(* IEC 61131-3 sources: myCodes/Stone/07.02.2022 - OOPs Approach/MPx_One_New/Mpx_One_Source_Code/MPx_One/3. USHPXMPX010A1/USHPXMPX010A1/[8c990d04-4ef8-4ca1-9757-e845a4517aeb]/Application, 12 files *)

(* ---- 010_GeneralMng.st ---- *)
USING System.UI;
USING System;
USING System.Timer;
USING System.Serial;
USING System.NVRAM;
USING System.Logs;
USING Libs.Blackout;
USING Libs.Logics;
USING System.Math;
USING System.Text;
USING libs.GenericFunctionMng;

{IF DEF(MPX_LOGS)}
(* ONLY FOR DEBUG *)
VAR_GLOBAL
	LogsBuffer : ARRAY [0..1024] OF BYTE;
    myStrDebugCarel : STRING;
END_VAR
(* -------------- *)
{ENDIF}

VAR_GLOBAL
    (**Detect restarts of MPXone application*)
    powerUp : BOOL;
    (**Flag for recognize that a defrost was performed*)
    DfrPerformed : BOOL;
    (**flag for save sw_version after RetainRestoreDefault()*)
    SW_Update    : BOOL;
    (* Backup BMS Configuration fo upgrade SW  ------*)
    BMS_Addr_bkp : USINT;
    BMS_Baud_bkp : USINT;
    BMS_Conf_bkp : USINT;
    BMS_Prot_bkp : BOOL;
END_VAR

VAR_GLOBAL RETAIN
    (**Number of restrts of MPXone application *)
    RestartsCounter : UINT;
END_VAR

VAR_GLOBAL PERSISTENT
    (**Start for periodic log: hour*)
    {METADATA MAX_VAL 23}
    {METADATA MIN_VAL 0}
    {ATTRIBUTE UOM HOUR}
    StartLog_Hour : USINT (0..23) := 0;
    (**Start for periodic log: minute*)
    {METADATA MAX_VAL 59}
    {METADATA MIN_VAL 0}
    {ATTRIBUTE UOM MINUTE}
    StartLog_Min : USINT (0..59) := 0;

    StartLog_DT : DATE_AND_TIME;
END_VAR

NAMESPACE LibraryNamespaceAndVersion

PROGRAM GeneralMng

    VAR
        BMS_BaudPrec, BMS_ConfPrec, BMS_AddrPrec : USINT;
        FB_BaudPrec : USINT;

        FirsCheckBlackout : BOOL := FALSE;
        BlackoutCtl : Blackout;
        MyLastOffDate : DATE_AND_TIME;
        NVRAM_Array : DWORD;
        myPwrOffDate_NVRAM_BLKO : UDINT;

        CngCnfRT                : RF_TRIG;
        R_Trig_enNFC : R_TRIG;

        TON_WAIT_DOWNLOAD : TON;

        FirstRun : BOOL := TRUE;

        prevZoneHmi : BOOL;
        pCOType, boardType, machineType, hwCode : UINT;

        SPV_DT : DT;
        prevSPV_DT : DT := DATE_AND_TIME#2017-01-01-00:00:00;
        DisSpvUpdF_APP : BOOL;

        cfgId : SINT;
        cfgOk : BOOL;
        {IF NOT DEF(MPXONE_BASIC)}
        cfgName : STRING[16];
        {ELSE}
        cfgName : STRING[4];
        {ENDIF}
        UniqueId : LWORD;
    END_VAR

    VAR_TEMP
        ProdCode_HwID : USINT;
        ProdCode_ProdVers : USINT;
        tmp_Startlog : DateTime;
        tmp_CurrTime : DateTime;
        lastDfrTime_DWORD : DWORD;
        swVersion_tmp           : UINT;
    END_VAR

    {REGION HARDWARE INFO}
    GetHardwareDescription(HwDesc);
    GetModel(pCOType, boardType, machineType, hwCode);
    GetProductInfo(Product_Info);

    IF firstCycle THEN
        UniqueId := TO_LWORD(GetUniqueId());
        Split_UniqueId(UniqueId, UniqueID_SPV);

        {IF DEF(MPXONE_ADVANCED)}
        PwrSupplyFailure := FALSE;
        uConfig[9].mode_sel := 0; // U9 set as analog input to manageultracap control
        {ENDIF}

    END_IF;

    IF Product_Info.ProductCode <> '' THEN
        ProdCode_HwID := TO_USINT(MID(Product_Info.ProductCode, 2, 10));
        isPanelVersion := (ProdCode_HwID >= 5) AND (ProdCode_HwID <= 8);
        ProdCode_ProdVers := TO_USINT(MID(Product_Info.ProductCode, 1, 6));
        isCustomBasicRU := (ProdCode_ProdVers < 3) AND (ProdCode_HwID = 5);
        isProdBasicVersion := (ProdCode_ProdVers <= 4) AND (ProdCode_HwID <= 6);
    ELSE
        isPanelVersion := FALSE;
    END_IF;

    IF isCustomBasicRU THEN
        Ain_Types.Group1 := 1;
    END_IF;
    {ENDREGION}

    {REGION RESET TO DEFAULT IF SW VERSION IS DIFFERET OR MANUAL RESET}
                // Compose version variable for BMS and for reeset for update SW
    swVersion_tmp := __PROJ_VER_MAJOR__ * 1000 + __PROJ_VER_MINOR__ * 100 + __PROJ_VER_BUILD__;

    IF SW_Update THEN                   // at restart after RetainRestoreDefault() (below)
        swVersion := swVersion_tmp;     // save SW version
        SW_Update := FALSE;             // Stop reset time

            //Restore BMS settings only on change version (NOT on Manual Default request)
        IF NOT ResCarelSets THEN
            BMS_Addr :=BMS_Addr_bkp;
            BMS_Baud :=BMS_Baud_bkp;
            BMS_Conf :=BMS_Conf_bkp;
            BMS_Prot :=BMS_Prot_bkp;
        END_IF;

        DispMngInst.StartSync(DownloadDir#ACUtoHMI, FALSE); //Force param from ACU to NFC
        //RetainForceBackup();
        ResCarelSets := FALSE;
    END_IF;
    IF (swVersion <> swVersion_tmp AND NOT(SW_Update)) OR ResCarelSets THEN
        // Backup BMS configuration only
        BMS_Addr_bkp :=BMS_Addr;
        BMS_Baud_bkp :=BMS_Baud;
        BMS_Conf_bkp :=BMS_Conf;
        BMS_Prot_bkp :=BMS_Prot;
        RetainRestoreDefault(); //keep one program loop to be executed
        SW_Update    := TRUE;
    END_IF;
    {ENDREGION}

    {REGION Set DEFAULT values for analog input channels}

    // wiz done from Applica
    // for wiz done from HMI see: WIZ_ENDPRG.st
    IF WizDone AND WizProgress THEN
        WizDone_Action();
    END_IF;
    {ENDREGION}

    {REGION RESTART COUNTER}
    IF NOT powerUp THEN
        //poerUp := FALSE in PROGRAM OutputsMng
        RestartsCounter     := RestartsCounter + 1;
        LogsEventsCounter   := LogsEventsCounter + 1;
    END_IF;
    {ENDREGION}

    {REGION NFC and DISPLAY CHANGE management}
    R_Trig_enNFC(CLK := EnNfc);
    IF EnNfc THEN //AND NOT firstCycle THEN
        //DispMngInst.Check(isPanelVersion, IsCommissioningToolPresent() OR NOT(MasterOnlineTON.Q));
        IF NOT R_Trig_enNFC.Q OR NOT powerUp THEN
            DispMngInst.Check(FALSE, IsCommissioningToolPresent() OR NOT(MasterOnlineTON.Q));
        ELSE
            DispMngInst.StartSync(DownloadDir#ACUtoHMI, R_Trig_enNFC.Q);
        END_IF;

        //forcing parameter values from ACU to HMI in case of display change
        IF DispMngInst.isWaitingForUser() THEN
            NewDispPrompt := FALSE;
            DispMngInst.StartSync(DownloadDir#ACUtoHMI, FALSE);
        END_IF;
    END_IF;
    {ENDREGION}

    {IF DEF(NO_SEV_SUPPORT)}
	OneRow.Init();
	OneRow.Read();
    {ENDIF}

    // Find related compilation DEFINES
    {IF DEF(MPXONE_BASIC)}
    isBasic := TRUE;
    isMedium := FALSE;
    isAdvanced := FALSE;
    {ENDIF}

    {IF DEF(MPXONE_MEDIUM)}
    isBasic := TRUE;
    isMedium := TRUE;
    isAdvanced := FALSE;
    {ENDIF}

    {IF DEF(MPXONE_ADVANCED)}
    isBasic := TRUE;
    isMedium := TRUE;
    isAdvanced := TRUE;
    {ENDIF}

    {REGION CHANGE BMS SETTINGS}

    SpvTable.SerialPort.Settings.Channel := Serial_Channel#BMS1;
    (*change of BMS supervisor baudrate*)
    SpvTable.SerialPort.Settings.Speed := SetSerialSpeed(BMS_Baud);

    (*change of BMS supervisor settings*)
    SpvTable.SerialPort.Settings.Bits := 8;
    IF BMS_Conf > 5 THEN
        BMS_Conf := 0;
    END_IF;
    CASE BMS_Conf OF
        0:
            SpvTable.SerialPort.Settings.Parity := Serial_Parity#None;
            SpvTable.SerialPort.Settings.Stops := 1;
            (*8 NONE 1*)

        1:
            SpvTable.SerialPort.Settings.Parity := Serial_Parity#None;
            SpvTable.SerialPort.Settings.Stops := 2;
            (*8 NONE 2*)

        2:
            SpvTable.SerialPort.Settings.Parity := Serial_Parity#Even;
            SpvTable.SerialPort.Settings.Stops := 1;
            (*8 EVEN 1*)

        3:
            SpvTable.SerialPort.Settings.Parity := Serial_Parity#Even;
            SpvTable.SerialPort.Settings.Stops := 2;
            (*8 EVEN 2*)

        4:
            SpvTable.SerialPort.Settings.Parity := Serial_Parity#Odd;
            SpvTable.SerialPort.Settings.Stops := 1;
            (*8 ODD 1*)

        5:
            SpvTable.SerialPort.Settings.Parity := Serial_Parity#Odd;
            SpvTable.SerialPort.Settings.Stops := 2;
            (*8 ODD 2*)
    END_CASE;

    // Carel protocol works only at 19200 8n2
    IF NOT BMS_Prot AND ( BMS_Baud <> 4 OR BMS_Conf <> 1 ) THEN
        BMS_Baud := 4;
        BMS_Conf := 1;
    END_IF;

    (*change setting of supervisor port, just in case of modifications*)
    IF BMS_Baud <> BMS_BaudPrec OR BMS_Conf <> BMS_ConfPrec OR BMS_Addr <> BMS_AddrPrec THEN
        (* Set ID to allow STone communication *)
        SetModbusDebugID(BMS_Addr, SpvTable.serialPort.Settings.Channel);
        (* Adjust settings *)
        SerialChangeSettings(SpvTable.serialPort.Settings);

        IF BMS_Prot THEN
            MB_Slave.ChangeIdent(BMS_Addr);
        END_IF;

        BMS_BaudPrec := BMS_Baud;
        BMS_ConfPrec := BMS_Conf;
        BMS_AddrPrec := BMS_Addr;

        // Set the same settings for BMS port on Default app (In case of FW ugrade the device will be reachable with the same settings)
        SaveIdePortSettings(SpvTable.SerialPort.Settings.Channel, SpvTable.SerialPort.Settings.Speed,
            SpvTable.SerialPort.Settings.Bits, SpvTable.SerialPort.Settings.Parity, SpvTable.SerialPort.Settings.Stops, BMS_Addr);
    END_IF;

    IF FB_Baud <> FB_BaudPrec OR Fieldbus.SerialSettings.Speed <> SetSerialSpeed(FB_Baud) THEN

        Fieldbus.SerialSettings.Speed := SetSerialSpeed(FB_Baud);
        SerialChangeSettings(Fieldbus.SerialSettings);
        //Fieldbus.ChangeSettings();

        FB_BaudPrec := FB_Baud;
    END_IF;

    IF ZoneHMI THEN
        SpvTable.Info.Zone := System.Globalization.Imperial;
    ELSE
        SpvTable.Info.Zone := System.Globalization.SI;
    END_IF;

    IF ZoneHMI <> prevZoneHmi THEN
        prevZoneHmi := ZoneHMI;
        ChangedUoM := TRUE;
    ELSE
        ChangedUoM := FALSE;
    END_IF;

    Libs.SPV_Gateway_HPX.InitProtocols();

    IF WizDone AND NOT SlvUpdFW THEN

        SpvTable.Read(ChangedUoM, BMS_Prot);
        FieldBus.Read();
        {IF NOT DEF(NO_MPXONE_REPEATER)}
        mpxRepeater.Init(198, repeaterConfig);
        mpxRepeater.Check(HmiRemSel > 0);
        {ENDIF}
    END_IF;

    {ENDREGION }

    {REGION RTC WRITE}

    (*sets the time from app through NFC*)
    IF ToggleSetTimeAPP THEN

        SetTime(DateTimeToSet);
        SetTimeZone(Posix);

        // Avoid unexpected defrost changing RTC time
        GetLocalTime(CurrDateTime);
        //DfrStartedDT := CurrDateTime;

        ToggleSetTimeAPP := FALSE;
        //DisSpvUpdF := TRUE;
        DisSpvUpdF_APP := TRUE;

        // Reset alarm if any
        Alarms.Al.Al_RTC.Info.Trigger := FALSE;
    END_IF;

    // Update SPV Variables
    SPV_DT := CONCAT_DT(TO_UINT(SPV_Year) + 2000, TO_UINT(SPV_Month), TO_UINT(SPV_Day), TO_UINT(SPV_Hour), TO_UINT(SPV_Min), 0, 0);
    IF SPV_DT <> prevSPV_DT AND NOT FirstRun THEN

        // SPV has updated date/time of controller
        SetLocalTime(SPV_DT);

        // Avoid unexpected defrost changing RTC time
        GetLocalTime(CurrDateTime);
        //DfrStartedDT := CurrDateTime;

        // Reset alarm if any
        Alarms.Al.Al_RTC.Info.Trigger := FALSE;
    END_IF;
    prevSPV_DT := SPV_DT;

    (*return the local time of the control*)
    GetLocalTime(CurrDateTime);
    CurrentDoW := DAY_OF_WEEK(CurrDateTime);

    IF FirstRun THEN
        SPV_DoW := CurrentDoW;
        updateDateTimeVar(CurrDateTime, SPV_Day, SPV_Month, SPV_Year, SPV_Hour, SPV_Min);
        SPV_DT := CONCAT_DT(TO_UINT(SPV_Year) + 2000, TO_UINT(SPV_Month), TO_UINT(SPV_Day), TO_UINT(SPV_Hour), TO_UINT(SPV_Min), 0, 0);
        prevSPV_DT := SPV_DT;
    END_IF;

    // WARNING: Current Date
    // Normal time flow
    IF NOT DisSpvUpdF_APP THEN
        SPV_CurrDoW := TO_USINT(CurrentDoW);
        updateDateTimeVar(CurrDateTime, SPV_CurrDay, SPV_CurrMonth, SPV_Curryear, SPV_CurrHour, SPV_CurrMin);
//        SPLIT_DT(CurrDateTime, tmpYear, tmpMonth, tmpDay, tmpHour, tmpMin, tmpSec, tmpMillis);
//        SPV_CurrYear := TO_REAL(tmpYear - 2000);
//        SPV_CurrMonth := TO_REAL(tmpMonth);
//        SPV_CurrDay := TO_REAL(tmpDay);
//        SPV_CurrHour := TO_REAL(tmpHour);
//        SPV_CurrMin := TO_REAL(tmpMin);
    ELSE
        DisSpvUpdF_APP := FALSE;
    END_IF;

    IF NOT WizDone THEN
        Alarms.Al.Al_RTC.Info.Trigger := FALSE;
    END_IF;

    {ENDREGION}

    {REGION LOGS management}

    IF NOT FirstRun THEN

        SPLIT_DT(StartLog_DT, tmp_Startlog);
        IF ((StartLog_Hour <> 0) OR (StartLog_Min <> 0)) AND
            ((StartLog_Hour <> TO_USINT(tmp_Startlog.Hour)) OR (StartLog_Min <> TO_USINT(tmp_Startlog.Minute))) THEN

            SPLIT_DT(CurrDateTime, tmp_CurrTime);
            StartLog_DT := CONCAT_DT(tmp_CurrTime.Year, tmp_CurrTime.Month, tmp_CurrTime.Day,
                            TO_UINT(StartLog_Hour), TO_UINT(StartLog_Min), 0, 0);
        ELSIF (StartLog_DT > DT#2000-01-01-00:00:00) AND
            ((StartLog_Hour <> 0) OR (StartLog_Min <> 0))THEN
            IF (CurrDateTime >= StartLog_DT) THEN
                Logs.Check();
            END_IF;
        ELSE
            StartLog_DT := DT#2000-01-01-00:00:00;
        END_IF;
    END_IF;

//    IF SamplingTime > 0 THEN
//        RS_StartLogs(S := (StartLog_DT > T#0ms) AND (CurrTime_Logs >= StartLog_DT), R1 := StopPeriodicsLogs);

//        IF RS_StartLogs.Q1 THEN
//           AND ((CurrDateTime - prevCurrDateTime) >= TO_TIME(TO_UDINT(SamplingTime) * 3600 * 1000)) THEN
//            prevCurrDateTime := CurrDateTime;
//            LogsEventsCounter := LogsEventsCounter + 1;

//            IF DfrPerformedCntLog <> DfrPerformedCntLog_prev THEN
//                DfrPerformedCntLog_prev := DfrPerformedCntLog;
//                DfrPerformed := TRUE;
//            ELSE
//                DfrPerformed := FALSE;
//            END_IF;

    {ENDREGION}

    /* **************************************************************************************/
    /*                                                                                      */
    /* MPXone NVRAM STRUCTURE:                                                              */
    /* from byte 0 to byte 3 --> Blackout management                                        */
    /* from byte 4 to byte 7 --> Management of the saving of the last defrost starting      */
    /*                                                                                      */
    /* ************************************************************************************ */

    {REGION READ LAST DEFROST TIME}
    NVRAM_ReadVar(4, lastDfrTime_DWORD);
    IF lastDfrTime_DWORD <> 0 THEN
        DfrStartedDT := TO_DT(lastDfrTime_DWORD);
        IF CurrDateTime - DfrStartedDT < T#0h THEN //if different is out of range (too big)
            SetLastDfrTime_RTC_MEM(CurrDateTime);
        END_IF;
    END_IF;
    {ENDREGION}

    {REGION BLACKOUT}

//    CurrentDate_UDINT := TO_UDINT(CurrDateTime);
    IF NOT FirsCheckBlackout THEN
        //read
        NVRAM_ReadVar(0, NVRAM_Array);
        myPwrOffDate_NVRAM_BLKO := TO_UDINT(NVRAM_Array);
        FirsCheckBlackout := TRUE;
    ELSE
        NVRAM_Array := TO_DWORD(TO_UDINT(CurrDateTime));//TO_DWORD(CurrentDate_UDINT);
        NVRAM_WriteVar(0, NVRAM_Array);
        //read
        NVRAM_ReadVar(0, NVRAM_Array);
        myPwrOffDate_NVRAM_BLKO := TO_UDINT(NVRAM_Array);
    END_IF;
    BlackoutCtl(PwrOffDate_NVRAM_BLKO := myPwrOffDate_NVRAM_BLKO);
    MyLastOffDate := CONCAT_DT(BlackoutCtl.LastOnYear_BLKO,
                               BlackoutCtl.LastOnMonth_BLKO,
                               BlackoutCtl.LastOnDay_BLKO,
                               BlackoutCtl.LastOnHour_BLKO,
                               BlackoutCtl.LastOnMin_BLKO,
                               BlackoutCtl.LastOnSec_BLKO, 0);

    BlackoutSR(S1 := MyLastOffDate <> MyLastOffDate_Saved, R := NOT firstCycle);

    //IF MyLastOffDate_Saved > CurrDateTime THEN
    IF (CurrDateTime >= DT#1970-01-01-00:00:00) AND (CurrDateTime < DT#1970-01-02-00:00:00) THEN
        Alarms.Al.Al_RTC.Info.Trigger := TRUE;
    END_IF;

    MyLastOffDate_Saved := MyLastOffDate;

    {ENDREGION}

    {REGION SAFE DOWNLOAD}

    IF GetFullDownloadRequest() THEN (*catch the request of fulldownload*)
        // Close solenoid
        WaitForUpdate := TRUE; (*switch off the unit*)

        // Close EEV
        {IF NOT DEF(MPXONE_BASIC)}
        EnManExv := FALSE;
        MachineVars.ManualPositioner_vars.ManualPositioningEnable := TRUE;
        MachineVars.ManualPositioner_vars.ManualPositionSteps := 0;

        TON_WAIT_DOWNLOAD(IN := TRUE,PT := T#1s);
        IF MachineVars.Engine_vars.EEV_vars.CurrentEstimatedPosition = 0 AND NOT CompOn OR hwCode = 312 THEN // TODO Verify that 312 is only PC symulator
            //UnitStatus := FALSE; (*switch off the unit*)
            /*IF Info_PWRP.Info_RotorSpeed_Perc = 0 THEN
                (*when the compressor is off, the full download can be done*)
                SetIDESema(TO_INT(IDESEMA_FULLDOWNLOAD),TO_INT(SEMA_STATUS_GO));
            ELSE
                (*waiting the compressor switch off*)
                SetIDESema(TO_INT(IDESEMA_FULLDOWNLOAD),TO_INT(SEMA_STATUS_WAIT));
            END_IF;*/
            // Conferma
            SetIDESema(TO_INT(IDESEMA_FULLDOWNLOAD),TO_INT(SEMA_STATUS_GO));
        END_IF;
        {ENDIF}

        {IF NOT DEF(MPXONE_MEDIUM)}
        TON_WAIT_DOWNLOAD(IN := TRUE,PT := T#1s);
        IF NOT CompOn OR hwCode = 312 THEN // TODO Verify that 312 is only PC symulator
            //UnitStatus := FALSE; (*switch off the unit*)
            /*IF Info_PWRP.Info_RotorSpeed_Perc = 0 THEN
                (*when the compressor is off, the full download can be done*)
                SetIDESema(TO_INT(IDESEMA_FULLDOWNLOAD),TO_INT(SEMA_STATUS_GO));
            ELSE
                (*waiting the compressor switch off*)
                SetIDESema(TO_INT(IDESEMA_FULLDOWNLOAD),TO_INT(SEMA_STATUS_WAIT));
            END_IF;*/
            // Conferma
            SetIDESema(TO_INT(IDESEMA_FULLDOWNLOAD),TO_INT(SEMA_STATUS_GO));
        END_IF;
        {ENDIF}
    ELSE
        TON_WAIT_DOWNLOAD(IN := FALSE,PT := T#0s);
        SetIDESema(TO_INT(IDESEMA_FULLDOWNLOAD),TO_INT(SEMA_STATUS_WAIT));
        WaitForUpdate := FALSE; (*switch off the unit*)
    END_IF;

    {ENDREGION}

    {IF DEF(NO_SEV_SUPPORT)}
    Libs.ReportSlaveID.ReportSlaveID(OneRow.Info.ReportSlaveID, OneRow.GetID(), OneRow.Info.Zone);
	OneRow.Write();
    {ENDIF}

	(* Refresh UI *)
	SendVirtualKey(NO_KEY, 1);

    // Visual store configuration (APP) management
    IF FirstRun THEN

        // Prepare the controller to store log messages
        {IF DEF(MPX_LOGS)}InitLog(LogsBuffer);{ENDIF}

        IF DfrStartedDT <= DT#1970-01-01-00:00:00 THEN
            DfrStartedDT := CurrDateTime;
        END_IF;

        // Reset the quick commands retained in NFC

        FirstRun := FALSE;
    END_IF;

    // Passthrough timeout
    PassThroughTON(IN := SlvUpdFW, PT := T#30s);
    IF PassThroughTON.Q THEN
        SlvUpdFW := FALSE;
    END_IF;

    // Configuration lookup
    //FOR cfgId := 0 TO 6 DO
        cfgOk := GetConfigurationName(TO_USINT(cfgId), cfgName);
    //END_FOR;

    // Change config by DI
    CngCnfRT(CLK := DigitalInputs.Fct.Config);
    IF CngCnfRT.Q AND NOT firstCycle THEN
        IF DigitalInputs.Fct.Config THEN
            cfgOk := SetConfiguration('C1');
        ELSE
            cfgOk := SetConfiguration('C2');
        END_IF;
        cfgOk := cfgOk;
    END_IF;

    // Applica profile recognition
    isUser := TRUE;
    isService := TRUE;
    isManufacturer := TRUE;
END_PROGRAM

FUNCTION_BLOCK StoreConfigSave
    VAR_IN_OUT
        ExtConfig : ARRAY[*] OF USINT;
        Config : ARRAY[*] OF WORD;
    END_VAR
    VAR
        index, ArrayOffset : DINT;
        tmpVal : WORD;
    END_VAR

    FOR ArrayOffset := 0 TO UPPER_BOUND(Config, 1) DO
    	Config[ArrayOffset] := 0;
    	FOR	index := 0 TO 7 DO
    		IF index + ArrayOffset * 8 <= UPPER_BOUND(ExtConfig, 1) THEN
    			tmpVal := SHL(TO_WORD(ExtConfig[index + ArrayOffset * 8]), index * 2);
    			Config[ArrayOffset] := TO_WORD(Config[ArrayOffset]) OR tmpVal;
    		END_IF;
    	END_FOR;
    END_FOR;

END_FUNCTION_BLOCK

FUNCTION_BLOCK StoreConfigRead
    VAR_IN_OUT
        ExtConfig : ARRAY[*] OF USINT;
        Config : ARRAY[*] OF WORD;
    END_VAR
    VAR
        index, ArrayOffset : DINT;
        tmpVal : WORD;
    END_VAR

    FOR ArrayOffset := 0 TO UPPER_BOUND(Config, 1) DO
    	//Config[ArrayOffset] := 0;
    	FOR	index := 0 TO 7 DO
    		IF index + ArrayOffset * 8 <= UPPER_BOUND(ExtConfig, 1) THEN
    			tmpVal := SHR(TO_WORD(Config[ArrayOffset]), index * 2);
    			ExtConfig[index + ArrayOffset * 8] := TO_USINT(tmpVal AND 2#11);
    		END_IF;
    	END_FOR;
    END_FOR;

END_FUNCTION_BLOCK

FUNCTION SetSerialSpeed : UDINT
    VAR_INPUT
        Index : USINT;
    END_VAR
    CASE Index OF
        0: SetSerialSpeed :=1200;
        1: SetSerialSpeed :=2400;
        2: SetSerialSpeed :=4800;
        3: SetSerialSpeed :=9600;
        4: SetSerialSpeed :=19200;
        5: SetSerialSpeed :=38400;
        6: SetSerialSpeed :=57600;
        7: SetSerialSpeed :=115200;
        8: SetSerialSpeed :=375000;
    END_CASE;
END_FUNCTION

FUNCTION updateDateTimeVar
    VAR_IN_OUT CONSTANT
        varCurrDateTime : DATE_AND_TIME;
    END_VAR

    VAR_IN_OUT
        varDay, varMonth, varYear, varHour, varMin : USINT;
    END_VAR

    VAR
        tmpYear, tmpMonth, tmpDay, tmpHour, tmpMin, tmpSec, tmpMillis : UINT;
    END_VAR

    SPLIT_DT(varCurrDateTime, tmpYear, tmpMonth, tmpDay, tmpHour, tmpMin, tmpSec, tmpMillis);
    varYear := TO_USINT(tmpYear - 2000);
    varMonth := TO_USINT(tmpMonth);
    varDay := TO_USINT(tmpDay);
    varHour := TO_USINT(tmpHour);
    varMin := TO_USINT(tmpMin);
END_FUNCTION

FUNCTION updateDateTimeVar
    VAR_IN_OUT CONSTANT
        varCurrDateTime : DATE_AND_TIME;
    END_VAR

    VAR_IN_OUT
        varDay, varMonth, varYear, varHour, varMin : REAL;
    END_VAR

    VAR
        tmpYear, tmpMonth, tmpDay, tmpHour, tmpMin, tmpSec, tmpMillis : UINT;
    END_VAR

    SPLIT_DT(varCurrDateTime, tmpYear, tmpMonth, tmpDay, tmpHour, tmpMin, tmpSec, tmpMillis);
    varYear := TO_REAL(tmpYear - 2000);
    varMonth := TO_REAL(tmpMonth);
    varDay := TO_REAL(tmpDay);
    varHour := TO_REAL(tmpHour);
    varMin := TO_REAL(tmpMin);
END_FUNCTION

FUNCTION Split_UniqueId
    VAR_IN_OUT CONSTANT
        UniqueID : LWORD;
    END_VAR

    VAR_IN_OUT
        UniqueID_splitted : ARRAY[*] OF USINT;
    END_VAR

    VAR
        i : DINT;
    END_VAR

    FOR i := LOWER_BOUND(UniqueID_splitted,1) TO UPPER_BOUND(UniqueID_splitted,1) DO
        UniqueID_splitted[i] := TO_USINT(SHR(UniqueID, i * 8));
    END_FOR;

END_FUNCTION

    /**
        Set DfrStartedDT
        Store on NVRAM DfrStartedDT
    */
FUNCTION SetLastDfrTime_RTC_MEM
    VAR_INPUT
        LastDfrTime : DT;
    END_VAR

    DfrStartedDT := LastDfrTime;
    NVRAM.NVRAM_WriteVar(4, TO_DWORD(DfrStartedDT));
END_FUNCTION

END_NAMESPACE

(* ---- 015_UnitStatus.st ---- *)
USING System.Math;

{DEFINE IDE_VER_1 1}
{DEFINE IDE_VER_2 3}
{DEFINE IDE_VER_3 3871}
{DEFINE IDE_VER_4 17150}

NAMESPACE LibraryNamespaceAndVersion

PROGRAM UnitStatusMng
        //wait restore default
    IF SW_Update THEN
        RETURN;
    END_IF;

{REGION Unit On Off}
    {IF __EDITOR_VER_1__ >= IDE_VER_1 AND __EDITOR_VER_2__ >= IDE_VER_2 AND __EDITOR_VER_3__ >= IDE_VER_3 AND __EDITOR_VER_4__ >= IDE_VER_4}
    UnitOn :=   NOT OrSeriousAlrm
                AND SEL(En_SupervOnOff, TRUE, SupervOnOff)
                AND SEL(Din_Cfg.Fct.RemoteOff.Ch <> 0,TRUE, NOT DigitalInputs.Fct.RemoteOff)
                AND SEL(En_KeyboardOnOff, TRUE, KeyboardOnOff);
    {ELSE}
    UnitOn :=   NOT OrSeriousAlrm
                AND SEL(En_SupervOnOff, SupervOnOff, TRUE)
                AND SEL(Din_Cfg.Fct.RemoteOff.Ch <> 0, NOT DigitalInputs.Fct.RemoteOff, TRUE)
                AND SEL(En_KeyboardOnOff, KeyboardOnOff, TRUE);
    {ENDIF}
{ENDREGION}

{REGION Unit Status}
    IF DfrStatus = DFR_DFR THEN
        UnitStatus := UNIT_STATUS#DEFROST;
    ELSIF ManContinuous THEN
        UnitStatus := UNIT_STATUS#CONTINUOS_CYCLE;
    ELSIF DutySettings THEN
        UnitStatus := UNIT_STATUS#DUTY_SETTINGS;
    ELSIF DigitalInputs.Fct.DoorOff OR DigitalInputs.Fct.DoorOn THEN
        UnitStatus := UNIT_STATUS#DOOR_OPEN;
    ELSIF ManClean THEN
        UnitStatus := UNIT_STATUS#CLEAN;
    ELSIF Alarms.Al.Status_Standby.Info.Active THEN
        UnitStatus := UNIT_STATUS#STANDBY;
    ELSIF En_KeyboardOnOff AND NOT KeyboardOnOff THEN
        UnitStatus := UNIT_STATUS#OFF_BY_KEYBOARD;
    ELSIF Din_Cfg.Fct.RemoteOff.Ch <> 0 AND DigitalInputs.Fct.RemoteOff THEN
        UnitStatus := UNIT_STATUS#OFF_BY_DIGITAL_INPUT;
    ELSIF En_SupervOnOff AND NOT SupervOnOff THEN
        UnitStatus := UNIT_STATUS#OFF_BY_SUPERVISOR;
    ELSIF OrSeriousAlrm THEN
        UnitStatus := UNIT_STATUS#OFF_BY_ALARM;
    ELSE
        UnitStatus := UNIT_STATUS#UNIT_ON;
    END_IF;
{ENDREGION}

{REGION UNIT STATUS WORKING MODE}
    CASE UnitStatus OF
        UNIT_STATUS#OFF_BY_ALARM,
        UNIT_STATUS#OFF_BY_DIGITAL_INPUT,
        UNIT_STATUS#OFF_BY_KEYBOARD,
        UNIT_STATUS#OFF_BY_SUPERVISOR,
        UNIT_STATUS#OFF_BY_TIME_BAND:
            {IF __EDITOR_VER_1__ >= IDE_VER_1 AND __EDITOR_VER_2__ >= IDE_VER_2 AND __EDITOR_VER_3__ >= IDE_VER_3 AND __EDITOR_VER_4__ >= IDE_VER_4}
            UnitStatus_WorkingMode := SEL(OrAlrm, UNIT_STATUS_GEN_FCT#UNIT_OFF, UNIT_STATUS_GEN_FCT#UNIT_ALARM);
            {ELSE}
            UnitStatus_WorkingMode := SEL(OrAlrm, UNIT_STATUS_GEN_FCT#UNIT_ALARM, UNIT_STATUS_GEN_FCT#UNIT_OFF);
            {ENDIF}
        UNIT_STATUS#UNIT_ON:
            {IF __EDITOR_VER_1__ >= IDE_VER_1 AND __EDITOR_VER_2__ >= IDE_VER_2 AND __EDITOR_VER_3__ >= IDE_VER_3 AND __EDITOR_VER_4__ >= IDE_VER_4}
            UnitStatus_WorkingMode := SEL(TempRegStatus, UNIT_STATUS_GEN_FCT#UNIT_ON, UNIT_STATUS_GEN_FCT#REGULATION_ON);
            {ELSE}
            IF OrAlrm THEN
                UnitStatus_WorkingMode := UNIT_STATUS_GEN_FCT#UNIT_ALARM;
            ELSIF TempRegStatus THEN
                UnitStatus_WorkingMode := UNIT_STATUS_GEN_FCT#REGULATION_ON;
            ELSE
                UnitStatus_WorkingMode := UNIT_STATUS_GEN_FCT#UNIT_ON;
            END_IF;
            {ENDIF}
        UNIT_STATUS#DEFROST:
            UnitStatus_WorkingMode := UNIT_STATUS_GEN_FCT#DEFROST;
        UNIT_STATUS#CLEAN:
            UnitStatus_WorkingMode := UNIT_STATUS_GEN_FCT#CASE_CLEANING;
        UNIT_STATUS#CONTINUOS_CYCLE:
            UnitStatus_WorkingMode := UNIT_STATUS_GEN_FCT#CONT_CYCLE;
        UNIT_STATUS#DUTY_SETTINGS:
            UnitStatus_WorkingMode := UNIT_STATUS_GEN_FCT#DUTY_SETTINGS;
        UNIT_STATUS#STANDBY:
            UnitStatus_WorkingMode := UNIT_STATUS_GEN_FCT#STANDBY;
        UNIT_STATUS#DOOR_OPEN:
            UnitStatus_WorkingMode := UNIT_STATUS_GEN_FCT#DOOR_OPEN;
        ELSE
            {IF __EDITOR_VER_1__ >= IDE_VER_1 AND __EDITOR_VER_2__ >= IDE_VER_2 AND __EDITOR_VER_3__ >= IDE_VER_3 AND __EDITOR_VER_4__ >= IDE_VER_4}
            UnitStatus_WorkingMode := SEL(OrAlrm, UNIT_STATUS_GEN_FCT#UNKNOWN, UNIT_STATUS_GEN_FCT#UNIT_ALARM);
            {ELSE}
            UnitStatus_WorkingMode := SEL(OrAlrm, UNIT_STATUS_GEN_FCT#UNIT_ALARM, UNIT_STATUS_GEN_FCT#UNKNOWN);
            {ENDIF}
    END_CASE;
{ENDREGION}

END_PROGRAM

END_NAMESPACE

(* ---- 020_InputsMng.st ---- *)
USING System.IO;
USING Libs.CustomGas;
USING System;
USING System.Timer;
USING System.Math;
USING Libs.Gas_GetCoeff;
USING Libs.Thermodynamic;
USING Libs.IOMng_Basic;

NAMESPACE LibraryNamespaceAndVersion

PROGRAM InputsMng
    VAR
        firstCycle_Local : BOOL := TRUE;

        TON_SerialBackup : TON;
        TON_SerialTimeout : ARRAY [1..4] OF TON;

        //Al_PrbBroken : ARRAY [1..PRB_NUM] OF Alarm.AlarmInfo;
        Al_SerialInputs : ARRAY [1..SER_AIN] OF Alarm.AlarmInfo;

        Sint : REAL;

        Simulation: ARRAY [1..MAX_AIN] OF PrbSimulation;
        F_TRIG_Simulation : F_TRIG;
        //SimVal : ARRAY [1..MAX_AIN] OF REAL;
        {IF NOT DEF(MPXONE_BASIC)}
        Coeff_PressToTemp : ARRAY[1..6] OF REAL;
        {ENDIF}

        EvapPBroken : BOOL := FALSE;

    END_VAR

    VAR_TEMP
        i : DINT;
        SerialAinIsUsed : ARRAY[1..4] OF BOOL;
        Ain_Max         : AinUnion;
        Ain_Min         : AinUnion;
        AinGroupCfg_arr : ARRAY [1..5]   OF MPX_AinGroupCfg;
    END_VAR

        //wait restore default
    IF SW_Update THEN
        RETURN;
    END_IF;

    {REGION PARAMETERS_TO_ARRAYS}
    IF NOT powerUp THEN
        //Reset probe settings
        FOR i := 1 TO TO_DINT(MAX_AIN_CH) DO
            uConfig[i].filter       := 5;
            uConfig[i].mode_sel     := LIB_IO_PIN_NOT_CONFIGURED;
            uConfig[i].mode_type    := LIB_IO_PROBE_NO_CONN;
        END_FOR;
    END_IF;
    {ENDREGION }

    {REGION START_UP_INPUT}
    IF firstCycle_Local THEN
        REPEATerConfig.CommandDelay := 2;
        REPEATerConfig.DetectionTimeOut := 500;
        REPEATerConfig.TimeOut := 500;

        (*this procedure is done every on*)
        firstCycle_Local := FALSE;
    END_IF;
    {ENDREGION }

    {REGION I/O configuration}
    // Convert active probe limits to union
    Ain_Max.Fct.EvapP := EvapMax;
    Ain_Min.Fct.EvapP := EvapMin;
    Ain_Max.Fct.AmbientH    := AmbHMax;
    Ain_Min.Fct.AmbientH    := AmbHMin;

    //Assign Probe group types
    AinGroupCfg_arr[1].ModeType := GetChannelType(Ain_Types.Group1);
{IF NOT DEF(MPXONE_BASIC)}
    AinGroupCfg_arr[2].ModeType := GetChannelType(Ain_Types.Group2);
    AinGroupCfg_arr[3].ModeType := GetChannelType(Ain_Types.Group3);
{ENDIF}
    {IF DEF(MPXONE_ADVANCED)}
    AinGroupCfg_arr[4].ModeType := GetChannelType(Ain_Types.Group4);
    AinGroupCfg_arr[5].ModeType := GetChannelType(Ain_Types.Group5);
    {ENDIF}

    //Set probe stability
    AinGroupCfg_arr[1].Filter := MAX(TO_USINT(TO_LREAL(AinStability) / 1.5), 1);
    AinGroupCfg_arr[2].Filter := MAX(TO_USINT(TO_LREAL(AinStability) / 1.5), 1);
    AinGroupCfg_arr[3].Filter := MAX(TO_USINT(TO_LREAL(AinStability) / 1.5), 1);

    FOR i := LOWER_BOUND(Ain_Cfg.Arr,1) TO UPPER_BOUND(Ain_Cfg.Arr,1) DO
        CASE Ain_Cfg.Arr[i].Ch OF
            0:
                Ain_Cfg.Arr[i].ModeType := Libs.IOMng_Basic.MODE_TYPE_AIN#LIB_IO_PROBE_NO_CONN;
                Ain_Cfg.Arr[i].Filter := 9;
            1,2,3:
                Ain_Cfg.Arr[i].ModeType := AinGroupCfg_arr[1].ModeType;
                Ain_Cfg.Arr[i].Filter := AinGroupCfg_arr[1].Filter;
            4,5:
                Ain_Cfg.Arr[i].ModeType := AinGroupCfg_arr[2].ModeType;
                Ain_Cfg.Arr[i].Filter := AinGroupCfg_arr[2].Filter;
            6:
                Ain_Cfg.Arr[i].ModeType := AinGroupCfg_arr[3].ModeType;
                Ain_Cfg.Arr[i].Filter := AinGroupCfg_arr[3].Filter;
            {IF DEF(MPXONE_ADVANCED)}
            7:
                Ain_Cfg.Arr[i].ModeType := AinGroupCfg_arr[4].ModeType;
                Ain_Cfg.Arr[i].Filter := AinGroupCfg_arr[4].Filter;
            8:
                Ain_Cfg.Arr[i].ModeType := AinGroupCfg_arr[5].ModeType;
                Ain_Cfg.Arr[i].Filter := AinGroupCfg_arr[5].Filter;
            {ENDIF}
        END_CASE;

        Ain_Cfg.Arr[i].Enable := Ain_Cfg.Arr[i].Ch <> 0;
        Ain_Cfg.Arr[i].AlrmDT := 0;//10; replace when new LibIO_mng will be ready 28/09/2020

    END_FOR;

    FOR i := LOWER_BOUND(Din_Cfg.Arr,1) TO UPPER_BOUND(Din_Cfg.Arr,1) DO
        Din_Cfg.Arr[i].Enable := Din_Cfg.Arr[i].Ch <> 0;
    END_FOR;

    FOR i := LOWER_BOUND(Dout_Cfg.Arr,1) TO UPPER_BOUND(Dout_Cfg.Arr,1) DO
            DOut_Cfg.Arr[i].Enable := DOut_Cfg.Arr[i].Ch <> 0;
    END_FOR;
    {ENDREGION}

    {REGION Ain simulated values}
    // Calc simulation data
    F_TRIG_Simulation(CLK := SimulateMode);

    IF SimulateMode THEN
        FOR i := LOWER_BOUND(Simulation, 1) TO UPPER_BOUND(Simulation, 1) DO
            Simulation[i].Config(SimMin[i], SimMax[i], SimPeriod[i]);
            virtU[i] := TRUE;
            U[i].r := Simulation[i].Run();
        END_FOR;
    END_IF;
    IF F_TRIG_Simulation.Q THEN
        FOR i := LOWER_BOUND(virtU, 1) TO UPPER_BOUND(virtU, 1) DO
            virtU[i] := FALSE;
        END_FOR;
    END_IF;
    {ENDREGION}

    {REGION PROBE_READING}
    // Clear alarms for unused input
    FOR i := LOWER_BOUND(Alarms.Al.Al_PrbBroken, 1) TO UPPER_BOUND(Alarms.Al.Al_PrbBroken, 1) DO
        Alarms.Al.Al_PrbBroken[i].Info.Trigger := FALSE;
    END_FOR;

    IO_mng.Read(
        0,
        ID,
        U,
        Din_Cfg.Arr,
        Ain_Cfg.Arr,
        Ain_Max.Arr,
        Ain_Min.Arr,
        Ain_offset.arr,
        DigitalInputs.Arr,
        Din_Err.Arr,
        AnalogInputs.Arr,
        Ain_Err.Arr,
        uConfig
        );

            // serial probe --------------------------------------------------
    FOR i :=1 TO UPPER_BOUND(Ain_Cfg.Arr,1) DO
        IF Ain_Cfg.Arr[i].Ch < 0 AND Ain_Cfg.Arr[i].Ch >= -4  THEN
            AnalogInputs.Arr[i] := SerialInputs[-Ain_Cfg.Arr[i].Ch].r;
            SerialAinIsUsed[- Ain_Cfg.Arr[i].Ch] := TRUE;
        END_IF;
    END_FOR;

    // Loop all AIN function block
    FOR i := LOWER_BOUND(AnalogInputs.Arr, 1) TO UPPER_BOUND(AnalogInputs.Arr, 1) DO
        IF TO_DINT(Ain_Cfg.Arr[i].Ch) >= LOWER_BOUND(Alarms.Al.Al_PrbBroken, 1) AND TO_DINT(Ain_Cfg.Arr[i].Ch) <= UPPER_BOUND(Alarms.Al.Al_PrbBroken, 1) THEN
            Alarms.Al.Al_PrbBroken[Ain_Cfg.Arr[i].Ch].Info.Trigger := Ain_Err.Arr[i].Trigger;
        END_IF;
    END_FOR;

    //Pressure probe alarm management during defrost [d12]
    IF (DfrStatus > DFR_IDLE AND DfrStatus < DFR_POST_DRIPPING) AND
        (Ain_Cfg.Fct.EvapP.Ch > 0 AND TO_DINT(Ain_Cfg.Fct.EvapP.Ch) <= UPPER_BOUND(Alarms.Al.Al_PrbBroken, 1)) THEN
        Alarms.Al.Al_PrbBroken[Ain_Cfg.Fct.EvapP.Ch].Info.Trigger := Alarms.Al.Al_PrbBroken[Ain_Cfg.Fct.EvapP.Ch].Info.Trigger AND (DfrPrbAlm <> 0 AND DfrPrbAlm <> 2);
    END_IF;

{IF NOT DEF(MPXONE_BASIC)}
    //ONLY FOR DATA LOG PURPOSE
    IF ((Ain_Cfg.Fct.EvapP.ch >= 1 AND Ain_Cfg.Fct.EvapP.ch <= 3) AND Ain_Types.Group1 = 1) OR
        ((Ain_Cfg.Fct.EvapP.ch >= 4 AND Ain_Cfg.Fct.EvapP.ch <= 5) AND Ain_Types.Group2 = 1) OR
        (Ain_Cfg.Fct.EvapP.ch = 6 AND Ain_Types.Group3 = 1) THEN

        EvapTempNTC_Log := AnalogInputs.Fct.EvapP;
        AnalogInputs.Fct.EvapP := 0.0;
    END_IF;
{ENDIF}
    {ENDREGION }

    {REGION UPDATE SLAVES PROBE}
    IF isMaster THEN
        FOR i := 1 TO TO_DINT(SlavesNum) DO
            {IF NOT DEF(MPXONE_BASIC)}
            Slaves[i].myHoldingRegisters[213] := TO_UINT(EvapSatTemp * 10.0);
            Slaves[i].myHoldingRegisters[214] := TO_UINT(AnalogInputs.Fct.EvapP * 10.0);
            Slaves[i].myHoldingRegisters[215] := TO_UINT(AnalogInputs.Fct.AmbientH * 10.0);
            Slaves[i].myHoldingRegisters[216] := TO_UINT(AnalogInputs.Fct.AmbientT * 10.0);
            Slaves[i].myHoldingRegisters[217] := TO_UINT(AnalogInputs.Fct.DewPoint * 10.0);
            {ELSE}
            Slaves[i].myHoldingRegisters[017] := TO_UINT(AnalogInputs.Fct.AmbientH * 10.0);
            Slaves[i].myHoldingRegisters[016] := TO_UINT(AnalogInputs.Fct.AmbientT * 10.0);
            Slaves[i].myHoldingRegisters[018] := TO_UINT(AnalogInputs.Fct.DewPoint * 10.0);
            {ENDIF}
        END_FOR;
    ELSE
        // For unconfigured probe on slave take value from master
        {IF NOT DEF(MPXONE_BASIC)}
        IF Ain_Cfg.Fct.EvapP.Ch = 0 THEN AnalogInputs.Fct.EvapP := MstEvapP; EvapSatTemp := MstEvapSatTemp; END_IF;
        {ELSE}
        IF Ain_Cfg.Fct.EvapP.Ch = 0 THEN (*AnalogInputs.Fct.EvapP := MstEvapP;*) EvapSatTemp := MstEvapSatTemp; END_IF;
        {ENDIF}
        IF Ain_Cfg.Fct.AmbientH.Ch = 0 THEN AnalogInputs.Fct.AmbientH := MstAmbientH; END_IF;
        IF Ain_Cfg.Fct.AmbientT.Ch = 0 THEN AnalogInputs.Fct.AmbientT := MstAmbientT; END_IF;
        IF Ain_Cfg.Fct.DewPoint.Ch = 0 THEN AnalogInputs.Fct.DewPoint := MstDewPoint; END_IF;

    END_IF;
    {ENDREGION}

    {REGION LOCAL_CONVERSION}
    // Local DewPoint conversion
    IF  NOT (Ain_Cfg.Fct.DewPoint.ch > 0) AND isMaster AND Ain_Cfg.Fct.AmbientT.ch <> 0 AND Ain_Cfg.Fct.AmbientH.ch <> 0 THEN
        IF AnalogInputs.Fct.AmbientT + 273.15 >0 THEN //èrotyect from negativbe logatithm
            AnalogInputs.Fct.DewPoint := DewPoint(AnalogInputs.Fct.AmbientT, AnalogInputs.Fct.AmbientH);
        END_IF;
    END_IF;

    // Glass probe estimate
    IF NOT (Ain_Cfg.Fct.GlassT.ch <> 0) THEN
        Sint := (AnalogInputs.Fct.AirOff * (100.0 - TO_REAL(GlassEstimComp)) + AnalogInputs.Fct.AirOn * TO_REAL(GlassEstimComp)) / 100;
        AnalogInputs.Fct.GlassT := (AnalogInputs.Fct.AmbientT - GlassTEstimateA) - (TO_REAL(GlassTEstimateB) / 100.0) *
            ((AnalogInputs.Fct.AmbientT - GlassTEstimateA) - Sint);
    END_IF;

    {IF NOT DEF(MPXONE_BASIC)}
    // Saturated temperature conversion
    IF RfrgTyp > 0 THEN
        Coeff_PressToTemp := GetCoeff_PressToTemp(TO_USINT(RfrgTyp - 1), ENUM_GAS_STATE#Dew);
        Alarms.Al.Al_GPE.Info.Active := FALSE;
    ELSE
        Alarms.Al.Al_GPE.Info.Active := NOT CheckCRC(CustomGasCoeff);
        Coeff_PressToTemp := ExtGasCoeff(CustomGasCoeff);
    END_IF;
    //Warning if no suction pressure probe configured
    Alarms.Al.Warn_SuctP_Prb.Info.Trigger := (ValveCnf = 1 OR ValveCnf = 2) AND Ain_Cfg.Fct.EvapP.ch = 0 AND isMaster;
    {ENDIF}

     // Suction pressure probe control lookup
    IF Ain_Cfg.Fct.EvapP.ch > 0 AND Ain_Cfg.Fct.EvapP.ch <= TO_SINT(MAX_AIN_CH) THEN
        EvapPBroken := Alarms.Al.Al_PrbBroken[Ain_Cfg.Fct.EvapP.ch].Info.Active;
    ELSIF Ain_Cfg.Fct.EvapP.ch < 0 AND Ain_Cfg.Fct.EvapP.ch >= -4 THEN
        EvapPBroken := Alarms.Al.Al_SerialInputs[-Ain_Cfg.Fct.EvapP.ch].Info.Active;
    ELSE
        // Probe not configured
        EvapPBroken := FALSE;
    END_IF;

    // Suction temperature probe control lookup
    IF Ain_Cfg.Fct.SuctT.ch > 0 AND Ain_Cfg.Fct.SuctT.ch <= TO_SINT(MAX_AIN_CH) THEN
        SuctTBroken := Alarms.Al.Al_PrbBroken[Ain_Cfg.Fct.SuctT.ch].Info.Active;
    ELSIF Ain_Cfg.Fct.SuctT.ch < 0 AND Ain_Cfg.Fct.SuctT.ch >= -4 THEN
        SuctTBroken := Alarms.Al.Al_SerialInputs[-Ain_Cfg.Fct.SuctT.ch].Info.Active;
    ELSE
        // Probe not configured
        SuctTBroken := FALSE;
    END_IF;

    //Backup value (P15) is used when: unit is master and the suctP probe is not configured or in alarm
    //                                 unit is slave suctP probe is not configured and communication is lost with master
    //                                 unit is slave suctP probe is not configured and suctP value is less or equal to zero (probe in alarm or not configured on master)
    //                                 unit is slave suctP probe IS configured locally and suctP probe is in alarm
    {IF NOT DEF(MPXONE_BASIC)}
    IF (IsMaster AND (Ain_Cfg.Fct.EvapP.ch = 0 OR EvapPBroken)) OR
        (Alarms.Al.Al_MA.Info.Active AND (Ain_Cfg.Fct.EvapP.ch = 0)) OR
        (NOT isMaster AND (Ain_Cfg.Fct.EvapP.ch = 0 AND AnalogInputs.Fct.EvapP <= 0) OR
                          (NOT (Ain_Cfg.Fct.EvapP.ch = 0) AND EvapPBroken)) THEN

        IF ValveCnf <> 6 THEN
            EvapSatTemp := ExvSatTempBackup;
        END_IF;

    ELSE
        EvapSatTemp := PressToTemp(AnalogInputs.Fct.EvapP, Coeff_PressToTemp) + EvapOffset;
    END_IF;
    {ENDIF}

    //tGS value in case of Suct Temp on Evd driver (ValveCnf = 6)
    {IF NOT DEF(MPXONE_BASIC)}
    IF ValveCnf = 6 THEN // P1 parameter
       AnalogInputs.Fct.SuctT := MachineVars.SH_vars.SuctionTemperature;
        AnalogInputs.Fct.EvapP := EVD_EvapP;
    END_IF;
    {ENDIF}

    // Copy all the values in common array for UI and Alarms
    FOR i := LOWER_BOUND(AnalogInputs.Arr, 1) TO UPPER_BOUND(AnalogInputs.Arr, 1) DO
        RegValues[i] := AnalogInputs.Arr[i];
    END_FOR;
    // Add the other value useful
    RegValues[AIN_NUM + 1] := VirtualProbe;
    RegValues[AIN_NUM + 2] := EvapSatTemp;
    {IF NOT DEF(MPXONE_BASIC)}
    RegValues[AIN_NUM + 3] := ActualSH;
    RegValues[AIN_NUM + 4] := TO_REAL(ExvVlvPosition);
    {ELIF NOT DEF(MPXONE_MEDIUM)}
    RegValues[AIN_NUM + 3] := 0.0;
    RegValues[AIN_NUM + 4] := 0.0;
    {ENDIF}
    RegValues[AIN_NUM + 5] := FansReq;
    RegValues[AIN_NUM + 6] := TO_REAL(HeatersOut);
    // !! TO ADD MORE VALUES INCREASE THE "EXTRA_VALUES" DEFINE VALUE !!

    {ENDREGION }

    {REGION DIGITAL_INPUT}
    // Virtual Digital Input
    FOR i := LOWER_BOUND(DigitalInputs.Arr, 1) TO UPPER_BOUND(DigitalInputs.Arr, 1) DO
        IF Din_Cfg.Arr[i].Ch = -1 THEN
            DigitalInputs.Arr[i] := VirtualDI;
        END_IF;
    END_FOR;

    // Digital input propagation from master to slave
    IF isMaster AND VirtualDiOut <> 0 THEN
        // set VirtualDI
        FOR i := 1 TO TO_DINT(SlavesNum) DO
            {IF NOT DEF(MPXONE_BASIC)}
            CASE VirtualDiOut OF
                -1 : Slaves[i].myCoilStatus[76] := VirtualDI;
                1..5 : Slaves[i].myCoilStatus[76] := ID[VirtualDiOut];
            END_CASE;
            {ELSE}
            CASE VirtualDiOut OF
                -1 : Slaves[i].myCoilStatus[068] := VirtualDI;
                1..5 : Slaves[i].myCoilStatus[068] := ID[VirtualDiOut];
            END_CASE;
            {ENDIF}

        END_FOR;
    END_IF;

    {ENDREGION}

    {REGION SERIAL_PROBE_BACKUP}
    // Restore at startup
    IF firstCycle_Local THEN
        SerialInputs := BakSerialInputs;
    END_IF;

    // Save every 30 minutes
    TON_SerialBackup(
        IN := NOT TON_SerialBackup.Q,
        PT := T#30m
        );
    IF TON_SerialBackup.Q THEN
        BakSerialInputs := SerialInputs;
    END_IF;

    FOR i := 1 TO 4 DO
        // Serial value timeout at 20 minutes
        TON_SerialTimeout[i](
            IN := (BakSerialInputs[i] = SerialInputs[i]) AND SerialAinIsUsed[i],
            PT := T#20m);

        Al_SerialInputs[i].Trigger := TON_SerialTimeout[i].Q;

    END_FOR;

    {ENDREGION}

    firstCycle_Local := FALSE;

END_PROGRAM

FUNCTION GetChannelType : USINT
    VAR_INPUT
        AinChannel : USINT;
    END_VAR

    CASE AinChannel OF
        0: //PT1000
            GetChannelType := libs.IOMng_Basic.MODE_TYPE_AIN#LIB_IO_PROBE_PT1000;
        1: //NTC
            GetChannelType := libs.IOMng_Basic.MODE_TYPE_AIN#LIB_IO_PROBE_NTC;
        2: //0-5V
            GetChannelType := libs.IOMng_Basic.MODE_TYPE_AIN#LIB_IO_PROBE_0_5V;
        3: //4-20mA
            GetChannelType := libs.IOMng_Basic.MODE_TYPE_AIN#LIB_IO_PROBE_4_20MA;
        4: //0-10V
            GetChannelType := libs.IOMng_Basic.MODE_TYPE_AIN#LIB_IO_PROBE_0_10V;
        5: //NTC-HT
            GetChannelType := libs.IOMng_Basic.MODE_TYPE_AIN#LIB_IO_PROBE_NTC_0_150;
        6: //0.5..4.5V
            GetChannelType := libs.IOMng_Basic.MODE_TYPE_AIN#LIB_IO_PROBE_05_45V;
    ELSE
        GetChannelType := AinChannel;
    END_CASE;

END_FUNCTION

CLASS PrbSimulation
    VAR
        Min: REAL := 0.0;
        Max: REAL := 100.0;
        Period : TIME := T#5m;
        {METADATA HIDDEN}
        counterP : TON;
        {METADATA HIDDEN}
        degrees : REAL;
    END_VAR

    METHOD Config
        VAR_INPUT
            Min: REAL;
            Max: REAL;
            Period : TIME;
        END_VAR

        THIS.Min := Min;
        THIS.Max := Max;
        THIS.Period := Period;
    END_METHOD

    METHOD Run : REAL

        IF Period <= T#0s THEN
            RETURN;
        END_IF;

        counterP(IN := NOT counterP.Q, PT := Period);
        degrees := (TO_REAL(counterP.ET) / TO_REAL(Period)) * 3.14159 * 2 ;

        Run := (SIN(degrees) + 1) / 2 * (THIS.Max - THIS.Min) + THIS.Min;
    END_METHOD
END_CLASS

END_NAMESPACE

(* ---- 030_AlarmsMng.st ---- *)
USING System;
USING System.Math;
USING System.Timer;
USING System.Alarm;
USING Libs.Alarm_Mng;
USING Libs.Hysteresis;

VAR_GLOBAL CONSTANT
    {IF NOT DEF(MPXONE_BASIC)}
    (**Global number of available alarms*)
    NUM_ALARMS : USINT := 56;
    (**Global number of available warning*)
    NUM_WARN_STATUS : USINT := 7;
    NUM_PRB_BROKEN : USINT := 8;
    {ELSE}
    (**Global number of available alarms*)
    NUM_ALARMS : USINT := 45;
    (**Global number of available warning*)
    NUM_WARN_STATUS : USINT := 5;
    NUM_PRB_BROKEN : USINT := 3;
    {ENDIF}
END_VAR

VAR_GLOBAL
    ActiveAlm : ARRAY[1..NUM_ALARMS + NUM_WARN_STATUS] OF UINT;
    //LstAlrmReq : ARRAY[1..NUM_ALARMS] OF Alarm_Req;
    Alarms : AlarmsUnion;
END_VAR

NAMESPACE LibraryNamespaceAndVersion

PROGRAM AlarmsMng
    VAR
        CleanLog : AlarmLog;
        //TON_AlrmResetDetect : TON;

        AlValue, Al2Value : REAL;
        //Alarm, Alarm2 : MpxAlarmMng;

        AlDinDelayTON : TON;

        ContCycleTON : TON;
        ContCycleF : F_EDGE;

        DfrTON : TON;
        DfrF : F_EDGE;

        HACCP_HA_TON : TON;

        ResetTON : TON;

        HACCP_LogTON : TON;

        DoorBypassTON : TON;
        DoorBypassRS : RS;

        (**Type HA & HF HACCP alarm*)
    	Al_HA, Al_HF : Alarm_Req := (Info := ( Code := 1, Category := 1));

        {IF NOT DEF(MPXONE_BASIC)}
        (**R_TRIG array for generate event log for probe broken and HI/Low tem alarms *)
        R_TRIG_AlarmsToLogEvent : ARRAY[1..8] OF R_TRIG;
        {ELSE}
        R_TRIG_AlarmsToLogEvent : ARRAY[1..5] OF R_TRIG;
        {ENDIF}

        HiAlarmThrTemp, HiAlarm2ThrTemp     : REAL;
        LowAlarmThrTemp, LowAlarm2ThrTemp   : REAL;

    END_VAR

    VAR_TEMP
        i : DINT;
        AlrmWord : WORD;
        //AlarmCodes : ARRAY [1..NUM_ALARMS] OF STRING[3];

        FakeReset : BOOL;
        ActiveHAAlarms, ActiveHFAlarms : ARRAY[0..2] OF UINT;
    END_VAR

    //wait restore default
    IF SW_Update THEN
        RETURN;
    END_IF;

    {REGION TEMPERATURE ALARM}

    // Fetch probe values for alarm management
    AlValue := ReadAlarmValue(AlarmPrbConf);
    Al2Value := ReadAlarmValue(Alarm2PrbConf);

    // Alarms are enabled?

    // Disable low alarm after continuous cycle
    ContCycleF(In := ManContinuous, Reset := ContCycleTON.Q);
    ContCycleTON(IN := ContCycleF.Out, PT := TO_TIME(TO_DINT(ContCycleLowBypass) * 60 * 1000));

    // Disable high alarm during dfr and in configured also after defrost
    DfrF(In := DfrStatus >= DFR_DFR, Reset := DfrTON.Q);
    DfrTON(IN := DfrF.Out, PT := TO_TIME(TO_DINT(DfrHiBypass) * 60 * 1000));
    DfrHiBypassEnd := DfrTON.Q;

    // Disable High temperature alarm during door open
    DoorBypassRS(S := DigitalInputs.Fct.DoorOn OR DigitalInputs.Fct.DoorOff, R1 := DoorBypassTON.Q OR NOT DoorBypassRS.S);
    DoorBypassTON(IN := DoorBypassRS.S, PT := TO_TIME(TO_DINT(AlBypassDoor) * 60 * 1000));

    IF AbsAlarmThr THEN //If absolute alarm
        HiAlarmThrTemp := HiAlarmThrAbs;     //AHA
        LowAlarmThrTemp := LowAlarmThrAbs;   //ALA
    ELSE
        HiAlarmThrTemp := HiAlarmThr;        //AH
        LowAlarmThrTemp := LowAlarmThr;      //AL
    END_IF;

    IF AbsAlarm2Thr THEN
        HiAlarm2ThrTemp := HiAlarm2ThrAbs;   //AHA2
        LowAlarm2ThrTemp := LowAlarm2ThrAbs; //ALA2
    ELSE
        HiAlarm2ThrTemp := HiAlarm2Thr;      //AH2
        LowAlarm2ThrTemp := LowAlarm2Thr;    //AL2
    END_IF;

    // Check alarm condition
    TempAlarms[1](Value := AlValue, Setpoint := TempSetP,
        HighThr := HiAlarmThrTemp, LowThr := LowAlarmThrTemp, Diff := AlarmResetDiff,
        Delay := AlarmDelay, Absolute := AbsAlarmThr, Reset := AlrmRes,
        DisHi := DoorBypassRS.Q1 OR DfrF.Out OR DfrStatus > DFR_IDLE,
        DisLow := ContCycleF.Out, Enable := UnitOn AND (AlarmPrbConf > 0));

    TempAlarms[2](Value := Al2Value, Setpoint := TempSetP2,
        HighThr := HiAlarm2ThrTemp, LowThr := LowAlarm2ThrTemp, Diff := AlarmResetDiff,
        Delay := Alarm2Delay, Absolute := AbsAlarm2Thr, Reset := AlrmRes,
        DisHi := (DoorBypassRS.Q1 OR DfrF.Out OR DfrStatus > DFR_IDLE),
        DisLow := ContCycleF.Out , Enable := UnitOn AND (Alarm2PrbConf > 0));

    // Trigger alarms if enabled and not during clean operation
    Alarms.Al.Al_HiTemp.Info.Trigger := TempAlarms[1].AlarmHi AND NOT Alarms.Al.Status_Clean.Info.Active;
    Alarms.Al.Al_LowTemp.Info.Trigger := TempAlarms[1].AlarmLow AND NOT Alarms.Al.Status_Clean.Info.Active;
    Alarms.Al.Al_HiTemp2.Info.Trigger := TempAlarms[2].AlarmHi AND NOT Alarms.Al.Status_Clean.Info.Active;
    Alarms.Al.Al_LowTemp2.Info.Trigger := TempAlarms[2].AlarmLow AND NOT Alarms.Al.Status_Clean.Info.Active;

    IF HACCP_AlrmDelay > 0 THEN
        // HACCP Alarm HA, high temperature during the operation
        HACCP_HA_TON(IN := TempAlarms[1].Hi, PT := TO_TIME((TO_DINT(HACCP_AlrmDelay) + TO_DINT(AlarmDelay)) * 60 * 1000));
        Al_HA.Info.Trigger := HACCP_HA_TON.Q;
        Al_HA( AlrmRes := FakeReset,
        	Lst_ActAlrm := ActiveHAAlarms,
        	Lst_LogAlrm := LogHACCP_HA,
        	Lst_LogAlrm_Idx := LogHACCP_HA_Index);

        HACCP_CountHA := 0;
        FOR i := LOWER_BOUND(LogHACCP_HA, 1) TO UPPER_BOUND(LogHACCP_HA, 1) DO
            IF LogHACCP_HA[i].Code > 0 THEN
                Alarms.Al.Al_HA.Info.Trigger := TRUE;
                HACCP_CountHA := HACCP_CountHA + 1;
            END_IF;
        END_FOR;

        // HACCP Alarm HF, high temperature after power failure (blackout)
        Al_HF.Info.Trigger := HACCP_AlrmDelay > 0 AND BlackoutSR.Q1 AND TempAlarms[1].Hi;
        Al_HF( AlrmRes := FakeReset,
        	Lst_ActAlrm := ActiveHFAlarms,
        	Lst_LogAlrm := LogHACCP_HF,
        	Lst_LogAlrm_Idx := LogHACCP_HF_Index);

        HACCP_CountHF := 0;
        FOR i := LOWER_BOUND(LogHACCP_HF, 1) TO UPPER_BOUND(LogHACCP_HF, 1) DO
            IF LogHACCP_HF[i].Code > 0 THEN
                Alarms.Al.Al_HF.Info.Trigger := TRUE;
                HACCP_CountHF := HACCP_CountHF + 1;
            END_IF;
        END_FOR;

    ELSE
        Alarms.Al.Al_HA.Info.Trigger := FALSE;
        Alarms.Al.Al_HF.Info.Trigger := FALSE;

        // Clear Logs
        LogHACCP_HA_Index := 0;
        LogHACCP_HF_Index := 0;
        FOR i := 1 TO TO_DINT(UPPER_BOUND(LogHACCP_HA, 1)) DO
            LogHACCP_HA[i] := CleanLog;
            LogHACCP_HF[i] := CleanLog;
        END_FOR;
    END_IF;

    // Wizard alarm inhibition
    IF NOT WizDone THEN
        FOR i := LOWER_BOUND(Alarms.Arr, 1) TO UPPER_BOUND(Alarms.Arr, 1) DO
            Alarms.Arr[i].Info.Trigger := FALSE;
            Alarms.Arr[i].Info.Active := FALSE;
        END_FOR;
    END_IF;

    // HACCP Log save
    HACCP_LogTON(IN := NOT HACCP_LogTON.Q, PT := HACCP_Period);
    IF HACCP_LogTON.Q THEN
        HACCP_LogBuffer[HACCP_LogIndex] := AlValue;

        HACCP_LogIndex := HACCP_LogIndex + 1;
        IF HACCP_LogIndex > TO_USINT(UPPER_BOUND(HACCP_LogBuffer,1)) THEN
            HACCP_LogIndex := TO_USINT(LOWER_BOUND(HACCP_LogBuffer, 1));
        END_IF;
    END_IF;

    {ENDREGION}

    {REGION DIGITAL INPUT ALARMS}
    // Immediate alarm (DIN)
    Alarms.Al.AlExtDin.Info.Trigger := DigitalInputs.Fct.Alarm;

    // Delayed alarm (DIN)
    AlDinDelayTON(IN := DigitalInputs.Fct.DelayedAl, PT := TO_TIME( TO_DINT(AlDinDelay) * 60 * 1000));
    Alarms.Al.AlDelayExtDin.Info.Trigger := AlDinDelayTON.Q;
    {ENDREGION}

    {REGION ALARM REQUEST}

    // Config probe broken alarms
    {IF NOT DEF(MPXONE_BASIC)}
    FOR i := 1 TO TO_DINT(MAX_AIN_ADVANCED) DO
        Alarms.Al.Al_PrbBroken[i].StrCode := ' E' + TO_STRING(i);
        Alarms.Al.Al_PrbBroken[i].Info.Category := PRB_ALARMS_TYPE;
    END_FOR;
    {ELSE}
    FOR i := 1 TO TO_DINT(MAX_AIN_BASIC) DO
        Alarms.Al.Al_PrbBroken[i].StrCode := ' E' + TO_STRING(i);
        Alarms.Al.Al_PrbBroken[i].Info.Category := PRB_ALARMS_TYPE;
    END_FOR;
    {ENDIF}

    // Serial probe alarms
    FOR i := 1 TO 4 DO
        Alarms.Al.Al_SerialInputs[i].StrCode := 'E1' + TO_STRING(i);
        Alarms.Al.Al_SerialInputs[i].Info.Category := PRB_ALARMS_TYPE;
    END_FOR;

    // Loop all the alarm array
    FOR i := LOWER_BOUND(Alarms.Arr, 1) TO UPPER_BOUND(Alarms.Arr, 1) DO
        Alarms.Arr[i].Info.Code := TO_UINT(i);
        Alarms.Arr[i](
            //StrCode := AlarmCodes[i],   // Insert the alarm code to display in mask
        	AlrmRes := AlrmRes,
        	Lst_ActAlrm := ActiveAlm,
        	Lst_LogAlrm := LogAlarms,
        	Lst_LogAlrm_Idx := LogAlrmIdx);
    END_FOR;

    // Alarm for slave devices when master is not polling
    MasterOnlineTON(IN := TRUE AND NOT IsDebuggerPresent(), PT := T#60s);
    Alarms.Al.Al_MA.Info.Trigger := MasterOnlineTON.Q AND NOT isMaster;

    // Loop the Communication error with Slave (only on Master) alarms
    FOR i := 1 TO TO_DINT(Libs.SPV_Gateway_HPX.MAX_SLAVES) DO
        Alarms.Al.Al_u[i].StrCode := 'u' + TO_STRING(i);
        Alarms.Al.Al_u[i].Info.Category := REG_ALARMS_TYPE;
        Alarms.Al.Al_u[i].Info.Trigger := NOT Slaves[i].Info.IsOnline AND SlavesNum >= TO_USINT(i) AND isMaster;
    END_FOR;

    // Loop the Alarm on unit 1 to 9 in the network
    FOR i := 1 TO TO_DINT(Libs.SPV_Gateway_HPX.MAX_SLAVES) DO
        Alarms.Al.Al_n[i].StrCode := 'n' + TO_STRING(i);
        IF SlaveAlarmCheck THEN
            Alarms.Al.Al_n[i].Info.Category := REG_ALARMS_TYPE;
        ELSE
            Alarms.Al.Al_n[i].Info.Category := 0;
        END_IF;
            // chech "OrAlrm" on Slaves
        {IF NOT DEF(MPXONE_BASIC)}
        Alarms.Al.Al_n[i].Info.Trigger := Slaves[i].Info.IsOnline AND Slaves[i].myInputStatus[67] AND SlavesNum >= TO_USINT(i) AND isMaster;
        {ELSE}
        Alarms.Al.Al_n[i].Info.Trigger := Slaves[i].Info.IsOnline AND Slaves[i].myInputStatus[055] AND SlavesNum >= TO_USINT(i) AND isMaster;
        {ENDIF}
    END_FOR;

    // Generic alarms
    Alarms.Al.Al_GHI_1.Info.Trigger := GenFctAlarm_Out[1].Hi;
    Alarms.Al.Al_GLO_1.Info.Trigger := GenFctAlarm_Out[1].Low;

    //Power failure alalrm
    {IF DEF (MPXONE_ADVANCED)}
    Alarms.Al.Al_Ultracap_EEV.Info.Trigger := PwrSupplyFailure;
    {ENDIF}

    {ENDREGION}

    {REGION CLEAR ALARMS LOG}
    IF LogAlrmRes THEN
        LogAlrmRes := FALSE;
        (*restart log*)
        LogAlrmIdx := 0;
        (*clear log list*)
        FOR i := 1 TO TO_DINT(UPPER_BOUND(LogAlarms, 1)) DO
            LogAlarms[i] := CleanLog;
        END_FOR;
    END_IF;
    {ENDREGION}

    {REGION ALARMS COUNT}
    AlrmWord := Alarm_Mng(ActiveAlm);
    OrWarning := AlrmWord.3;
    OrAlrm := AlrmWord.0 OR AlrmWord.1 OR AlrmWord.2;
    OrStatus := AlrmWord.4;
    OrPrbAlrm := AlrmWord.1;
    OrSeriousAlrm := FALSE;// AlrmWord.2; Set to FALSE because all the alarms have automatic reset

    (*COUNT TOTAL ALARM AND WARNING ACTIVE*)
    TotActAlm := 0;
    TotActWarning := 0;
    TotActStatus := 0;
    FOR i := LOWER_BOUND(ActiveAlm,1) TO TO_DINT(UPPER_BOUND(ActiveAlm, 1)) DO
        //IF ActiveAlm[i] >= CAT_ALARM THEN
        IF ActiveAlm[i] > 0 AND ActiveAlm[i] < REG_WARNINGS_TYPE THEN
            TotActAlm := TotActAlm + 1;
        END_IF;
        IF ActiveAlm[i] > 0 AND ActiveAlm[i] = REG_WARNINGS_TYPE THEN
            TotActWarning := TotActWarning + 1;
        END_IF;
        IF ActiveAlm[i] > 0 AND ActiveAlm[i] = REG_STATUS_TYPE THEN
            TotActStatus := TotActStatus + 1;
        END_IF;
    END_FOR;
    {ENDREGION}

    // On alarm reset keep it to TRUE for 3 seconds
    ResetTON(IN := AlrmRes, PT := T#3s);
    IF ResetTON.Q THEN
        AlrmRes := FALSE;
    END_IF;

    // During startup wizard and reset keep alarms output off
    IF NOT WizDone OR StartupReset OR firstCycle THEN
        OrWarning := FALSE;
        OrAlrm := FALSE;
        OrStatus := FALSE;
        TotActAlm := 0;
        TotActWarning := 0;
        TotActStatus := 0;
    END_IF;

    R_TRIG_AlarmsToLogEvent[1](CLK := Alarms.Al.Al_PrbBroken[1].Info.Trigger);
    R_TRIG_AlarmsToLogEvent[2](CLK := Alarms.Al.Al_PrbBroken[2].Info.Trigger);
    R_TRIG_AlarmsToLogEvent[3](CLK := Alarms.Al.Al_PrbBroken[3].Info.Trigger);
    {IF NOT DEF(MPXONE_BASIC)}
    R_TRIG_AlarmsToLogEvent[4](CLK := Alarms.Al.Al_PrbBroken[4].Info.Trigger);
    R_TRIG_AlarmsToLogEvent[5](CLK := Alarms.Al.Al_PrbBroken[5].Info.Trigger);
    R_TRIG_AlarmsToLogEvent[6](CLK := Alarms.Al.Al_PrbBroken[6].Info.Trigger);
    R_TRIG_AlarmsToLogEvent[7](CLK := Alarms.Al.Al_HiTemp.Info.Trigger);
    R_TRIG_AlarmsToLogEvent[8](CLK := Alarms.Al.Al_LowTemp.Info.Trigger);
    {ELSE}
    R_TRIG_AlarmsToLogEvent[4](CLK := Alarms.Al.Al_HiTemp.Info.Trigger);
    R_TRIG_AlarmsToLogEvent[5](CLK := Alarms.Al.Al_LowTemp.Info.Trigger);
    {ENDIF}

    FOR i := LOWER_BOUND(R_TRIG_AlarmsToLogEvent,1) TO UPPER_BOUND(R_TRIG_AlarmsToLogEvent,1) DO
        IF R_TRIG_AlarmsToLogEvent[i].Q THEN
            LogsEventsCounter := LogsEventsCounter + 1;
            IF DfrPerformedCntLog <> DfrPerformedCntLog_prev THEN
                DfrPerformedCntLog_prev := DfrPerformedCntLog;
                DfrPerformed := TRUE;
            ELSE
                DfrPerformed := FALSE;
            END_IF;
            EXIT;
        END_IF;
    END_FOR;

END_PROGRAM

FUNCTION_BLOCK MpxAlarmMng
    VAR_INPUT
        Value, Setpoint : REAL;
        HighThr, LowThr, Diff : REAL;

        Delay : USINT;
        Absolute : BOOL;
        Reset : BOOL;
        (** Disable high temperature alarm*)
        DisHi : BOOL;
        (** Disable low temperature alarm*)
        DisLow : BOOL;

        (** Global enable *)
        Enable : BOOL;
    END_VAR

    VAR_OUTPUT
        AlarmHi, AlarmLow : BOOL;
        Hi, Low : BOOL;
    END_VAR

    VAR
        HighHYST, LowHYST : HysterAdv;
        HighTON, LowTON : TON_PAUSE;
    END_VAR

    VAR_TEMP
        DisableHi, DisableLow : BOOL := FALSE;
    END_VAR;

    IF Enable THEN

        // Alarm disable in case of wrong input value
        IF Absolute THEN
            DisableHi := HighThr > 49.9 AND HighThr < 50.1;
            DisableLow := LowThr > -49.9 AND LowThr < -50.1;
        ELSE
            DisableHi := HighThr > -0.1 AND HighThr < 0.1;
            DisableLow := LowThr > -0.1 AND LowThr < 0.1;
        END_IF;

        // Alarm conditions
        IF Absolute THEN
//            HighHYST(In := Value, Left := HighThr - Diff, Right := HighThr, Reverse := FALSE);
            HighHYST(In := Value, SetP := HighThr, DiffLeft := Diff, DiffRight := 0.0, Reverse := FALSE);
//            LowHYST(In := Value, Left := LowThr, Right := LowThr + Diff, Reverse := TRUE);
            LowHYST(In := Value, SetP := LowThr, DiffLeft := 0.0, DiffRight := Diff, Reverse := TRUE);
        ELSE
//            HighHYST(In := Value, Left := HighThr - Diff + Setpoint, Right := HighThr + Setpoint, Reverse := FALSE);
            HighHYST(In := Value, SetP := HighThr + Setpoint, DiffLeft := Diff, DiffRight := 0.0, Reverse := FALSE);
//            LowHYST(In := Value, Left := Setpoint - LowThr, Right := Setpoint - LowThr + Diff, Reverse := TRUE);
            LowHYST(In := Value, SetP := Setpoint - LowThr, DiffLeft := 0.0, DiffRight := Diff, Reverse := TRUE);
        END_IF;

        // Alarm logic based on TON with the possibility of pause counter
        Hi := HighHYST.Out AND NOT DisableHi;
        Low := LowHYST.Out AND NOT DisableLow;

        // Alarm delay
        HighTON(IN := Hi AND NOT Reset/* AND NOT DisableHi*/, PAUSE := DisHi, PT := TO_TIME(TO_UDINT(Delay) * 60 * 1000));
        LowTON(IN := Low AND NOT Reset/* AND NOT DisableLow*/, PAUSE := DisLow, PT := TO_TIME(TO_UDINT(Delay) * 60 * 1000));

        // Alarm outut
        AlarmHi := HighTON.Q;
        AlarmLow := LowTON.Q;
    ELSE
        // Reset counters
        HighTON(IN := FALSE, PAUSE := FALSE, PT := TO_TIME(TO_UDINT(Delay) * 60 * 1000));
        LowTON(IN := FALSE, PAUSE := FALSE, PT := TO_TIME(TO_UDINT(Delay) * 60 * 1000));

        // Alarm output
        AlarmHi := HighTON.Q;
        AlarmLow := LowTON.Q;
    END_IF;

END_FUNCTION_BLOCK

FUNCTION ReadAlarmValue : REAL
    VAR_INPUT
        config : USINT;
    END_VAR
    // Default value
    ReadAlarmValue := 0;

    // Bound check
    IF config < TO_USINT(LOWER_BOUND(RegValues, 1)) OR
        config > TO_USINT(UPPER_BOUND(RegValues, 1)) THEN
        RETURN;
    END_IF;

    ReadAlarmValue := RegValues[config];

END_FUNCTION

(**
 *              TON_PAUSE - On-delay timing - state machine.
 *
 * Timer on delay supplies the input value IN at Q with a time delay when
 * a rising edge is detected at IN.
 * If input IN is only '1' for a short pulse(shorter than PT),
 * the timer is not started for this edge.
 *
 * @example
 *             +--------+        +---+   +-----------+
 *        IN   |        |        |   |   |           |
 *           --+        +--------+   +---+           +-------------
 *             t0       t1       t2  t3  t4          t7
 *                                          +--+
 *     PAUSE                                |  |
 *           -------------------------------+  +----------------
 *             t0       t1       t2  t3  t4 t5 t6
 *                  +---+                        +---+
 *        Q         |   |                        |   |
 *           -------+   +------------------------+   +-------------
 *               t0+PT  t1            t4+PT-(t6-t5)   t7
 *          PT      +---+                        +---+
 *           :     /    |            +          /    |
 *        ET :    /     |           /|      +--+     |
 *           :   /      |          / |     /         |
 *           :  /       |         /  |    /          |
 *           0-+        +--------+   +---+           +-------------
 *             t0       t1       t2  t3  t4          t7
 *
 *
 *         2        +---+                     +---+
 * STATE   1   +----+   |        +---+   +----+   |
 *         0 --+        +--------+   +---+        +------
 *)
FUNCTION_BLOCK TON_PAUSE
    VAR_INPUT
        (** Input variable of which to detect rising edge. *)
        IN : BOOL;
        (** Preset value (ms), duration of impulse Q. *)
        PT : TIME;
        (** Input variable to pause counter *)
        PAUSE : BOOL;
    END_VAR
    VAR_OUTPUT
        (** Impluse, his value become high if IN value is high at least for PT ms. *)
        Q : BOOL := FALSE;
        (** Current value of time (ms). *)
        ET : TIME := T#0s;
    END_VAR

    VAR
        MEM : UDINT;
        OLD_IN : BOOL;
        NORMA_CYCLE : BOOL;
    END_VAR

    IF NOT OLD_IN AND IN THEN
        Q := FALSE;
        MEM := GetSystemTime();
        ET := TO_TIME(0);
        NORMA_CYCLE := TRUE;
    END_IF;

    IF NORMA_CYCLE AND NOT PAUSE THEN
        IF ET < PT THEN
            ET := TO_TIME(GetSystemTime() - MEM);
        ELSE
            ET := PT;
            Q := TRUE;
        END_IF;
    END_IF;

    IF NORMA_CYCLE AND PAUSE THEN
        MEM := GetSystemTime() - TO_UDINT(ET);
    END_IF;

    IF OLD_IN AND NOT IN THEN
        Q := FALSE;
        ET := TO_TIME(0);
        NORMA_CYCLE := FALSE;
    END_IF;
    OLD_IN := IN;
END_FUNCTION_BLOCK

END_NAMESPACE

(* ---- 050_UnitStartUp.st ---- *)
NAMESPACE LibraryNamespaceAndVersion

PROGRAM UnitStartUpMng

    //wait restore default
    IF SW_Update THEN
        RETURN;
    END_IF;

    // At startup keep the regulation off
    StartupTimeTON(IN := firstCycle AND NOT StartupReset, PT := StartupTime);
    IF StartupTimeTON.Q THEN
        firstCycle := FALSE;
    END_IF;

    // Stop regolation
    IF StartupReset THEN
        firstCycle := TRUE;
    END_IF;

    // Display changed ?
    IF NewDispPrompt THEN
        firstCycle := TRUE;
    END_IF;

END_PROGRAM

END_NAMESPACE
